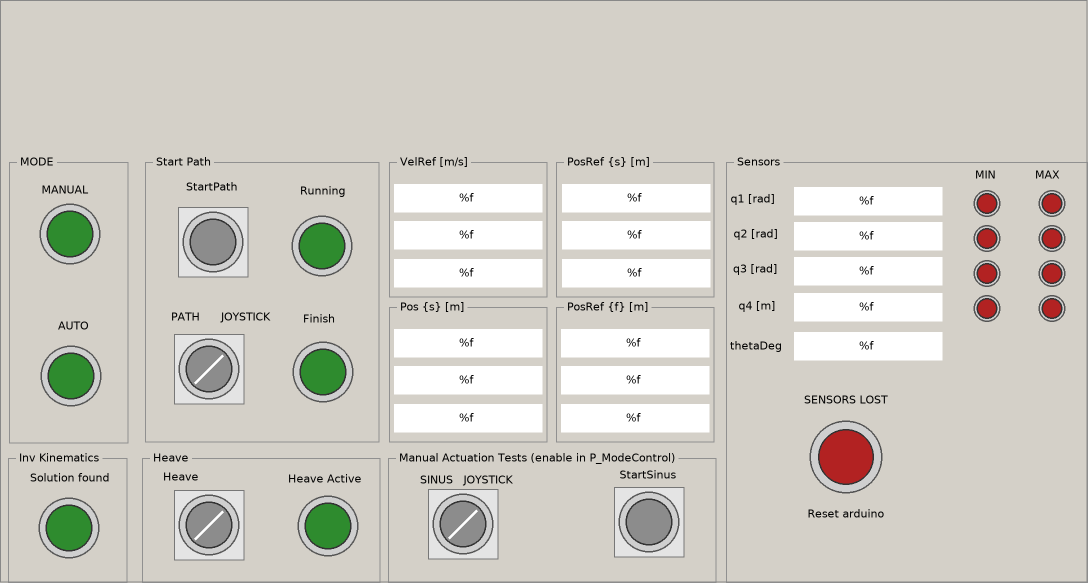
VISUALIZATION Visualization  // 1088x583
    GroupBox (388,450 328x133), "Manual Actuation Tests (enable in P_ModeControl)"
    GroupBox (389,154 158x143), "VelRef [m/s]"
        Label (99,258 150x30)
        Textfield (4,29 150x30), "%f", text variable: G_InverseKinematics.fvXref
        Textfield (4,66 150x30), "%f", text variable: G_InverseKinematics.fvYref
        Textfield (4,104 150x30), "%f", text variable: G_InverseKinematics.fvZref
    GroupBox (556,154 158x143), "PosRef {s} [m]"
        Textfield (5,29 150x30), "%f", text variable: G_Toolpoint.fXref
        Textfield (5,66 150x30), "%f", text variable: G_Toolpoint.fYref
        Textfield (5,104 150x30), "%f", text variable: G_Toolpoint.fZref
    GroupBox (389,299 158x143), "Pos {s} [m]"
        Textfield (4,29 150x30), "%f", text variable: G_Toolpoint.fX
        Textfield (4,66 150x30), "%f", text variable: G_Toolpoint.fY
        Textfield (4,104 150x30), "%f", text variable: G_Toolpoint.fZ
    GroupBox (9,154 119x289), "MODE"
        Lamp1 (26,45 70x70), variable: G_Buttons.bManualModeSelector, style: Lamp-Lamp1-Green
        Lamp1 (27,187 70x70), variable: G_Buttons.bAutoModeSelector, style: Lamp-Lamp1-Green
        Label (9,21 94x30), "MANUAL"
        Label (35,157 59x30), "AUTO"
    Label (113,154 150x30)
    GroupBox (145,154 234x288), "Start Path"
        Lamp1 (142,57 70x70), variable: G_Path.bPathRunning, style: Lamp-Lamp1-Green
        Lamp1 (143,183 70x70), variable: G_Path.bPathFinnish, style: Lamp-Lamp1-Green
        PushSwitch (33,53 70x70), variable: G_Path.bStartPath, behaviour: TOGGLE, style: Switch-PushSwitch-Gray
        Label (103,22 150x30), "Running"
        Label (99,150 150x30), "Finish"
        RotarySwitch (29,180 70x70), variable: G_Path.bPathActivated, behaviour: TOGGLE, style: Switch-RotarySwitch-Gray
        Label (7,148 137x30), "PATH JOYSTICK"
    Label (137,172 150x30), "StartPath"
    GroupBox (142,450 238x133), "Heave"
        Label (108,14 150x30), "Heave Active"
        RotarySwitch (32,40 70x70), variable: G_Heave.bHeaveEnable, behaviour: TOGGLE, style: Switch-RotarySwitch-Gray
        Lamp1 (151,41 70x70), variable: G_Heave.bHeaveActive, style: Lamp-Lamp1-Green
    Label (139,462 84x30), "Heave"
    GroupBox (8,450 119x133), "Inv Kinematics"
        Lamp1 (26,43 70x70), variable: G_InverseKinematics.bKinematicsSucsessful, style: Lamp-Lamp1-Green
        Label (16,13 92x30), "Solution found"
    GroupBox (726,154 362x429), "Sensors"
        Textfield (67,32 150x30), "%f", text variable: G_SensorsScaled.q1
        Textfield (67,67 150x30), "%f", text variable: G_SensorsScaled.q2
        Textfield (67,102 150x30), "%f", text variable: G_SensorsScaled.q3
        Textfield (67,138 150x30), "%f", text variable: G_SensorsScaled.q4
        Label (0,30 54x30), "q1 [rad]"
        Label (6,65 48x30), "q2 [rad]"
        Label (5,100 49x30), "q3 [rad]"
        Label (8,137 46x30), "q4 [m]"
        Label (104,181 150x30)
        Textfield (67,177 150x30), "%f", text variable: G_Heave.fTheta
        Label (0,177 60x30), "thetaDeg"
        Lamp1 (76,261 88x84), variable: G_SensorInput.bSensorDataLost, style: Lamp-Lamp1-Red
        Label (60,229 120x34), "SENSORS LOST"
        Label (60,343 120x34), "Reset arduino"
        Label (234,6 51x30), "MIN"
        Label (296,6 51x30), "MAX"
        Lamp1 (243,34 36x31), variable: G_ActuatorLimits.bq1Min, style: Lamp-Lamp1-Red
        Lamp1 (243,69 36x31), variable: G_ActuatorLimits.bq2Min, style: Lamp-Lamp1-Red
        Lamp1 (243,104 36x31), variable: G_ActuatorLimits.bq3Min, style: Lamp-Lamp1-Red
        Lamp1 (243,139 36x31), variable: G_ActuatorLimits.bq4Min, style: Lamp-Lamp1-Red
        Lamp1 (308,34 36x31), variable: G_ActuatorLimits.bq1Max, style: Lamp-Lamp1-Red
    Lamp1 (1034,223 36x31), variable: G_ActuatorLimits.bq2Max, style: Lamp-Lamp1-Red
    Lamp1 (1034,258 36x31), variable: G_ActuatorLimits.bq3Max, style: Lamp-Lamp1-Red
    Lamp1 (1034,293 36x31), variable: G_ActuatorLimits.bq4Max, style: Lamp-Lamp1-Red
    GroupBox (556,299 158x143), "PosRef {f} [m]"
        Textfield (4,29 150x30), "%f", text variable: G_Heave.r3x
        Textfield (4,66 150x30), "%f", text variable: G_Heave.r3y
        Textfield (4,104 150x30), "%f", text variable: G_Heave.r3z
    PushSwitch (614,487 70x70), variable: G_Servo.bStartSinus, behaviour: TOGGLE, style: Switch-PushSwitch-Gray
    Label (573,460 150x30), "StartSinus"
    RotarySwitch (428,489 70x70), variable: G_Servo.bSinusActive, behaviour: TOGGLE, style: Switch-RotarySwitch-Gray
    Label (398,465 137x30), "SINUS JOYSTICK"
END_VISUALIZATION

(* stored: Version 1.1.0.1, ProductVersion 3.1.4024.12
   Visu Visualization: Id {045ae3b7-7fee-47eb-a622-0401ba0fdac1} *)
